PROGRAM MAIN_FastAsPossible
VAR
	fbSetRtMode : FB_SetRtMode;
	fbGetRtMode : FB_GetRtMode;
	
	state : INT := 0;	
	bStart : BOOL; 
	iteration : INT := 0; 
END_VAR


VAR_OUTPUT 
	value AT %Q* : UDINT;	
END_VAR


fbSetRtMode(bExecute:=FALSE);
fbGetRtMode(bExecute:=FALSE);

CASE state OF
	0:
		IF(bStart = TRUE) THEN 		
			state:= 1;
			value:=100; // steps to decrement as Cyclic 
			iteration := iteration +1; 
		END_IF
	1:
		IF fbGetRtMode.bBusy = FALSE THEN  
			IF  fbGetRtMode.bError = FALSE  THEN
				IF fbGetRtMode.rtMode = E_RtMode.RtMode_Cyclic THEN
					state:=2; //if Cyclic start simulation = decremtn 
				ELSE
					fbGetRtMode(bExecute:= TRUE);
				END_IF
			ELSE	
				state:= 101;
			END_IF			
		END_IF
	2: 
		value:=value-1; //decrementing Cyclic (near realtime speed) 
		IF value = 0 THEN
			state := 3;
			fbSetRtMode(bExecute:= TRUE, rtMode:=E_RtMode.RtMode_FastAsPossible);			
		END_IF
	3:
		IF  fbSetRtMode.bBusy = FALSE THEN  
			IF fbSetRtMode.bError = FALSE THEN
				fbGetRtMode(bExecute:= TRUE);//querying RtMode  
				state := 4;
				value:=100000; // Steps to decrement as a FastAsPossible 						
			ELSE
				state := 101;
			END_IF  
		END_IF
	4:
		IF fbGetRtMode.bBusy = FALSE THEN  
			IF  fbGetRtMode.bError = FALSE  THEN
				IF fbGetRtMode.rtMode = E_RtMode.RtMode_FastAsPossible THEN
					state:=5; //if FastAsPossble start simulation = decremting 
				ELSE
					fbGetRtMode(bExecute:= TRUE);
				END_IF
			ELSE	
				state:= 102;
			END_IF			
		END_IF
	5: 
		value:=value-1; //decrementing as fast as possible 
		IF value = 0 THEN
			(*switch back to cyclic mode*)			
			fbSetRtMode(bExecute:= TRUE, rtMode:=E_RtMode.RtMode_Cyclic);
			state := 6;
		END_IF
	6:
		IF  fbSetRtMode.bBusy = FALSE THEN
			IF fbSetRtMode.bError = FALSE THEN
				state := 0;				
			ELSE
				state := 103;
			END_IF  
		END_IF	 	
END_CASE

END_PROGRAM

(* stored: Version 1.1.0.1, ProductVersion 3.1.4024.4
   POU MAIN_FastAsPossible: Id {9f632ce0-8bb6-426b-a741-962758f9f521}, SpecialFunc None *)
